{attribute 'GeneratedUsingTerminal: EP6224-0042-0016'}
{attribute addProperty BoxType "EP6224-0042-0016"}
{attribute addProperty Id "Digital_InputsDigital_Inputs_8749E1518"}
{attribute addProperty CRC "3668841627"}
{attribute addProperty Size "8"}
TYPE Module_7_Digital_Inputs_DAAE149B :
STRUCT
	{attribute addProperty Name "Digital_Inputs"}
	Digital_Inputs  : Digital_Inputs_8749E151;
END_STRUCT
END_TYPE

(* stored: Version 1.2.0.0, ProductVersion 3.1.4024.9
   DUT Module_7_Digital_Inputs_DAAE149B: Id {0a0452aa-c295-4184-b37e-5153b66bff96} *)
